FUNCTION_BLOCK FB_TrocarDetect
VAR_INPUT
END_VAR
VAR_OUTPUT
END_VAR
VAR
	m_trocarOnCounts :INT :=0;
	m_trocarOnCountThres :INT :=50;
END_VAR

// check if instrument is on
METHOD run : BOOL
VAR_INPUT
	IOValue :UDINT;
END_VAR
// trocar io is 5th bit 
IF 32=(IOValue AND 10#32) THEN
	m_trocarOnCounts :=MIN(m_trocarOnCounts +1,m_trocarOnCountThres);
ELSE
	m_trocarOnCounts :=0;
END_IF

run := m_trocarOnCounts >= m_trocarOnCountThres;
END_METHOD

END_FUNCTION_BLOCK

(* stored: Version 1.1.0.1, ProductVersion 3.1.4024.11
   POU FB_TrocarDetect: Id {c8d72a25-6879-4464-949d-51ce00faba6c}, SpecialFunc None
   Method run: Id {32b3fb7f-9cf2-40b4-b5e6-38652230a51d} *)
